FUNCTION_BLOCK ABSTRACT Button
VAR
	input AT %I* : BOOL;
END_VAR

PROPERTY PUBLIC State : BOOL
GET
state := input;
END_GET
END_PROPERTY

END_FUNCTION_BLOCK

(* stored: Version 1.1.0.1, ProductVersion 3.1.4024.12
   POU Button: Id {542591d4-41ca-44f4-bb69-3cd3f83d3355}, SpecialFunc None
   Property State: Id {c6b560a3-8daa-4eb4-b2d0-2c9676cc730e}
   Get Get: Id {660acae3-730e-4913-a5e7-94294b5faed6} *)
